FUNCTION Convert_STRING_TO_TOD : Hresult
VAR_INPUT
	in : STRING;
	out : REFERENCE TO TOD;
END_VAR
VAR
	converted : TOD;
END_VAR

converted := STRING_TO_TOD(in);

IF (TOD_TO_STRING(converted) <> in) THEN
	Convert_STRING_TO_TOD := INCOMPATIBLE;
	RETURN;
END_IF

out := converted;

END_FUNCTION

(* stored: Version 1.1.0.1, ProductVersion 3.1.4024.12
   POU Convert_STRING_TO_TOD: Id {da3b3560-9c72-4dc7-b658-00cc1f87f4dd}, SpecialFunc None *)
